PROGRAM P_StatusAnzeige
VAR
END_VAR

(*
Baustein: FC95 Status-Anzeige
Zeitstempel Code: 09.12.2014 10:56:48
Interface: 09.07.2010 10:27:01
*)

//NBT-NEU

GVL.zeigeFehler := (P_Ablauf.fbAllesInSollpos.bError AND NOT P_Ablauf.fbAllesInSollpos.bErrMute)
					OR P_FehlerAllgemein.fbKontrolleEndschalter.bError;


(* Netzwerk: 1 *)

//ToDo: Noch keine Ahnung, was das tun soll...
(*
L "DB6".d42 DB6.DBB42	-- Eingangs-Byte-Select Status

// https://www.sps-forum.de/simatic/81525-variabler-array-index-awl.html
//Beispiel:
//L #index    // 1..8 (aus MB23)
//+ -1        // --> 0..7
//SLD 3       // * 8 --> Byteadresse.0 -- Array_Index: 0 ... (muß * 8, weil Bit-Adressen adressiert werden, wir aber die Byte-Adresse brauchen)
			  //  Element_Größe: 1 = Byte / 2 = Word / 4 = DWord
			  

SLW 3 					-- Schiebt Wort um 3 bit nach links, bzw. multipliziert den Wert im Akku mit 8. Siehe oben...
// * 1 für Byte-Array rechnen nicht nötig

LAR1 					-- Akku als Zeiger in Adressregister 1 laden
L EB [AR1,P#0.0] 		-- Lade Eingangsbyte, Adressregister 1 mit Offset 0.0 adressiert
T "DB6".d40 DB6.DBB40 	-- 8*Eingangs-Bit Status
*)

(*
L "DB6".d46 DB6.DBB46 -- Ausgangs-Byte-Select Status
SLW 3
LAR1
L "DB6".d43 DB6.DBB43 -- Zuw.v.DBB46 Status
L "DB6".d46 DB6.DBB46 -- Ausgangs-Byte-Select Status
T "DB6".d43 DB6.DBB43 -- Zuw.v.DBB46 Status
==I
= L 0.0  -- L 0.0 ist das erste bit aus den lokaldaten
*)



(*
L "DB6".d45 DB6.DBB45 -- Zuw.vom selectierten Ausgangs-Byte Status
L AB [AR1,P#0.0]	  -- Lade Ausgangsbyte
T "DB6".d45 DB6.DBB45 -- Zuw.vom selectierten Ausgangs-Byte Status
<>I
R L 0.0
*)



(*
//https://www.sps-forum.de/simatic/6451-awl-anweisung-verstehen.html
//L 0.0 ist das erste bit aus den lokaldaten.
//Auf jeden Fall ist das keine saubere Arbeit. Siemens macht sowas gerne beim umschalten von KOP/FUP in AWL,
//aber ein Programmierer sollte das nicht tun.

U L 0.0
SPBN s1
*)

(*
	L "DB6".d44 DB6.DBB44 -- 8*Ausgangs-Bit Status
	T AB [AR1,P#0.0]
*)
	
(*	
s1: L AB [AR1,P#0.0]
	T "DB6".d44 DB6.DBB44 -- 8*Ausgangs-Bit Status
	L "DB6".d50 DB6.DBB50 -- Merker-Byte-Select Status
	SLW 3
	LAR1
	L "DB6".d47 DB6.DBB47 -- Zuw.v.DBB50 Status
	L "DB6".d50 DB6.DBB50 -- Merker-Byte-Select Status
	T "DB6".d47 DB6.DBB47 -- Zuw.v.DBB50 Status
	==I
	= L 0.0
	L "DB6".d49 DB6.DBB49 -- Zuw.vom selectierten Merker-Byte Status
	L MB [AR1,P#0.0]
	T "DB6".d49 DB6.DBB49 -- Zuw.vom selectierten Merker-Byte Status
	<>I
	R L 0.0
	U L 0.0
	SPBN s2
	L "DB6".d48 DB6.DBB48 -- 8*Merker-Bit Status
	T MB [AR1,P#0.0]
s2: L MB [AR1,P#0.0]
	T "DB6".d48 DB6.DBB48 -- 8*Merker-Bit Status
	L MW [AR1,P#0.0]
	T "DB6".d52 DB6.DBW52 -- Wert vom selectierten Merker-Byte Status
*)

;

END_PROGRAM

(* stored: Version 1.1.0.1, ProductVersion 3.1.4024.3
   POU P_StatusAnzeige: Id {320c13fb-4aa5-4aee-90d1-2a8f9646054a}, SpecialFunc None *)
